TYPE ST_OutputConvData :
STRUCT
	id :INT;
	timeStampin :STRING;
	timeStampout:STRING;
END_STRUCT
END_TYPE

(* stored: Version 1.1.0.1, ProductVersion 3.1.4026.17
   DUT ST_OutputConvData: Id {50cf2d9e-41c5-4bcf-ad34-f66d8ea3283e} *)
